PROGRAM AutoPreparationCtrl
VAR

	TON1: TON;
	TON2: TON;
	TON3: TON;
	TON4: TON;
	TON5: TON;
	TON6: TON;
	TON7: TON;
	TON8: TON;
	TON9: TON;
	TON10: TON;
	TON11: TON;
	TON12: TON;
	TON13: TON;
	TON14: TON;
	TON15: TON;
	TON16: TON;

	PreparationBypassTimer: TON;
	bPreparationBypassEn : BOOL;

	ARfbStnDegassCtrl: ARRAY [1..iStnQty] OF fbStnDegassCtrl;

	ARbStnDegassInProcess: ARRAY [1..iStnQty] OF BOOL;

	tStn1IncomingValveDelayOn: TON;
	tStn1aIncomingValveDelayOn: TON;
	tStn2IncomingValveDelayOn: TON;
	tStn3IncomingValveDelayOn: TON;
	tStn5IncomingValveDelayOn: TON;

	bA1PnpStep6: BOOL;
END_VAR
VAR // added by the converter: edge detectors and wires of the graphical bodies
    _w1 : BOOL;
END_VAR

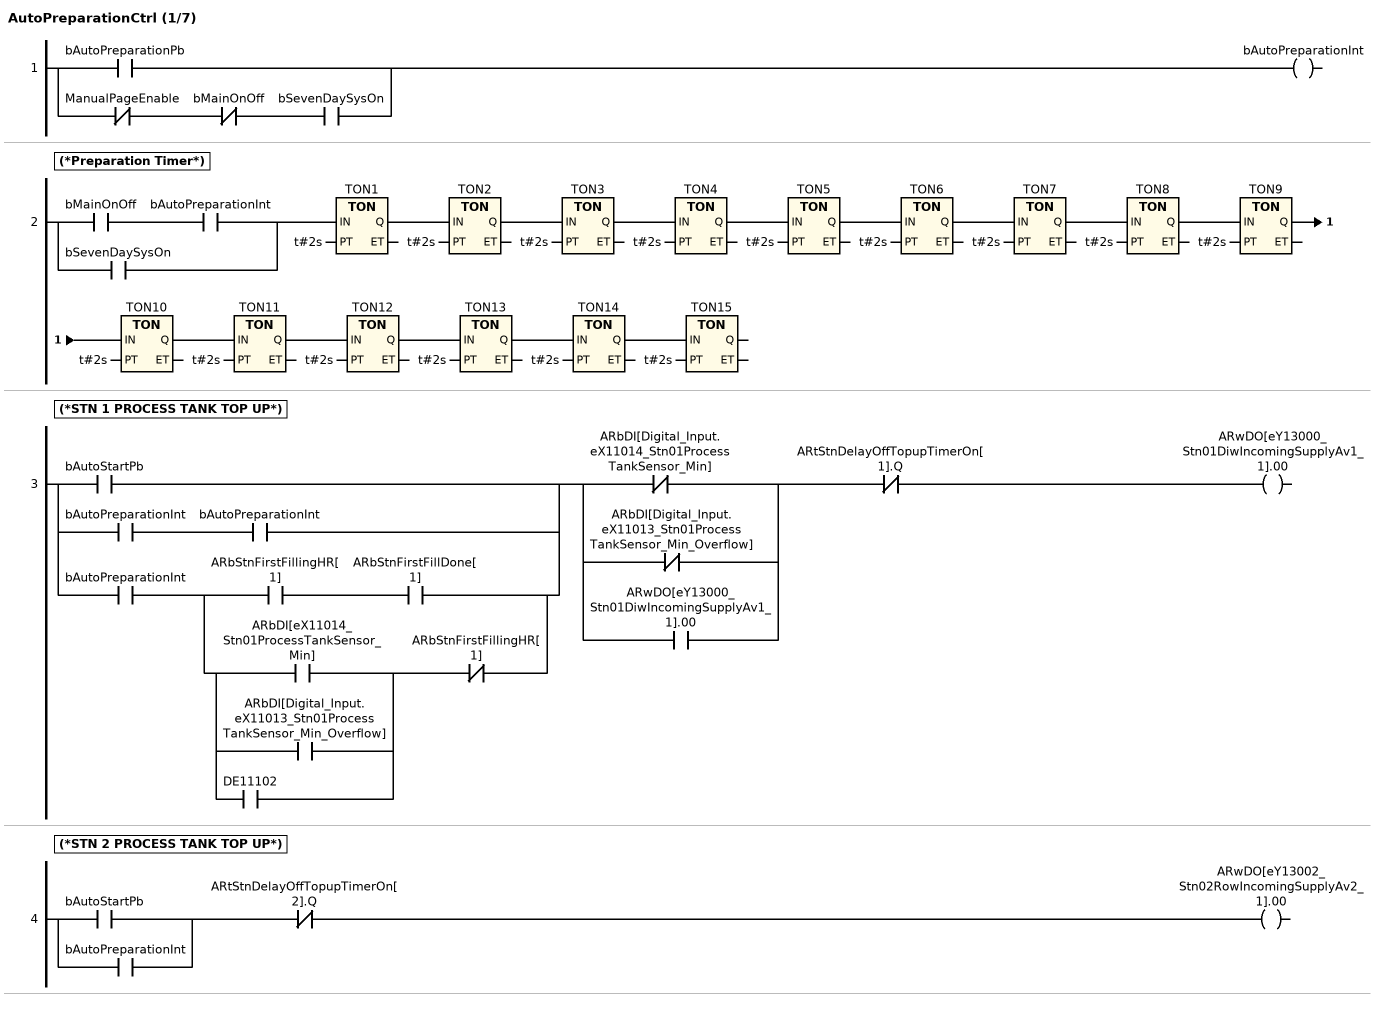
// NETWORK 1
bAutoPreparationInt := bAutoPreparationPb OR NOT ManualPageEnable AND NOT bMainOnOff AND bSevenDaySysOn;

// NETWORK 2
// label: (*Preparation Timer*)
TON1(IN := bMainOnOff AND bAutoPreparationInt OR bSevenDaySysOn, PT := t#2s); // TON
TON2(IN := TON1.Q, PT := t#2s); // TON
TON3(IN := TON2.Q, PT := t#2s); // TON
TON4(IN := TON3.Q, PT := t#2s); // TON
TON5(IN := TON4.Q, PT := t#2s); // TON
TON6(IN := TON5.Q, PT := t#2s); // TON
TON7(IN := TON6.Q, PT := t#2s); // TON
TON8(IN := TON7.Q, PT := t#2s); // TON
TON9(IN := TON8.Q, PT := t#2s); // TON
TON10(IN := TON9.Q, PT := t#2s); // TON
TON11(IN := TON10.Q, PT := t#2s); // TON
TON12(IN := TON11.Q, PT := t#2s); // TON
TON13(IN := TON12.Q, PT := t#2s); // TON
TON14(IN := TON13.Q, PT := t#2s); // TON
TON15(IN := TON14.Q, PT := t#2s); // TON

// NETWORK 3
// label: (*STN 1 PROCESS TANK TOP UP*)
ARwDO[eY13000_Stn01DiwIncomingSupplyAv1_1].00 := (bAutoStartPb OR bAutoPreparationInt AND bAutoPreparationInt OR bAutoPreparationInt AND (ARbStnFirstFillingHR[1] AND ARbStnFirstFillDone[1] OR (ARbDI[eX11014_Stn01ProcessTankSensor_Min] OR ARbDI[Digital_Input.eX11013_Stn01ProcessTankSensor_Min_Overflow] OR DE11102) AND NOT ARbStnFirstFillingHR[1])) AND (NOT ARbDI[Digital_Input.eX11014_Stn01ProcessTankSensor_Min] OR NOT ARbDI[Digital_Input.eX11013_Stn01ProcessTankSensor_Min_Overflow] OR ARwDO[eY13000_Stn01DiwIncomingSupplyAv1_1].00) AND NOT ARtStnDelayOffTopupTimerOn[1].Q;

// NETWORK 4
// label: (*STN 2 PROCESS TANK TOP UP*)
ARwDO[eY13002_Stn02RowIncomingSupplyAv2_1].00 := (bAutoStartPb OR bAutoPreparationInt) AND NOT ARtStnDelayOffTopupTimerOn[2].Q;

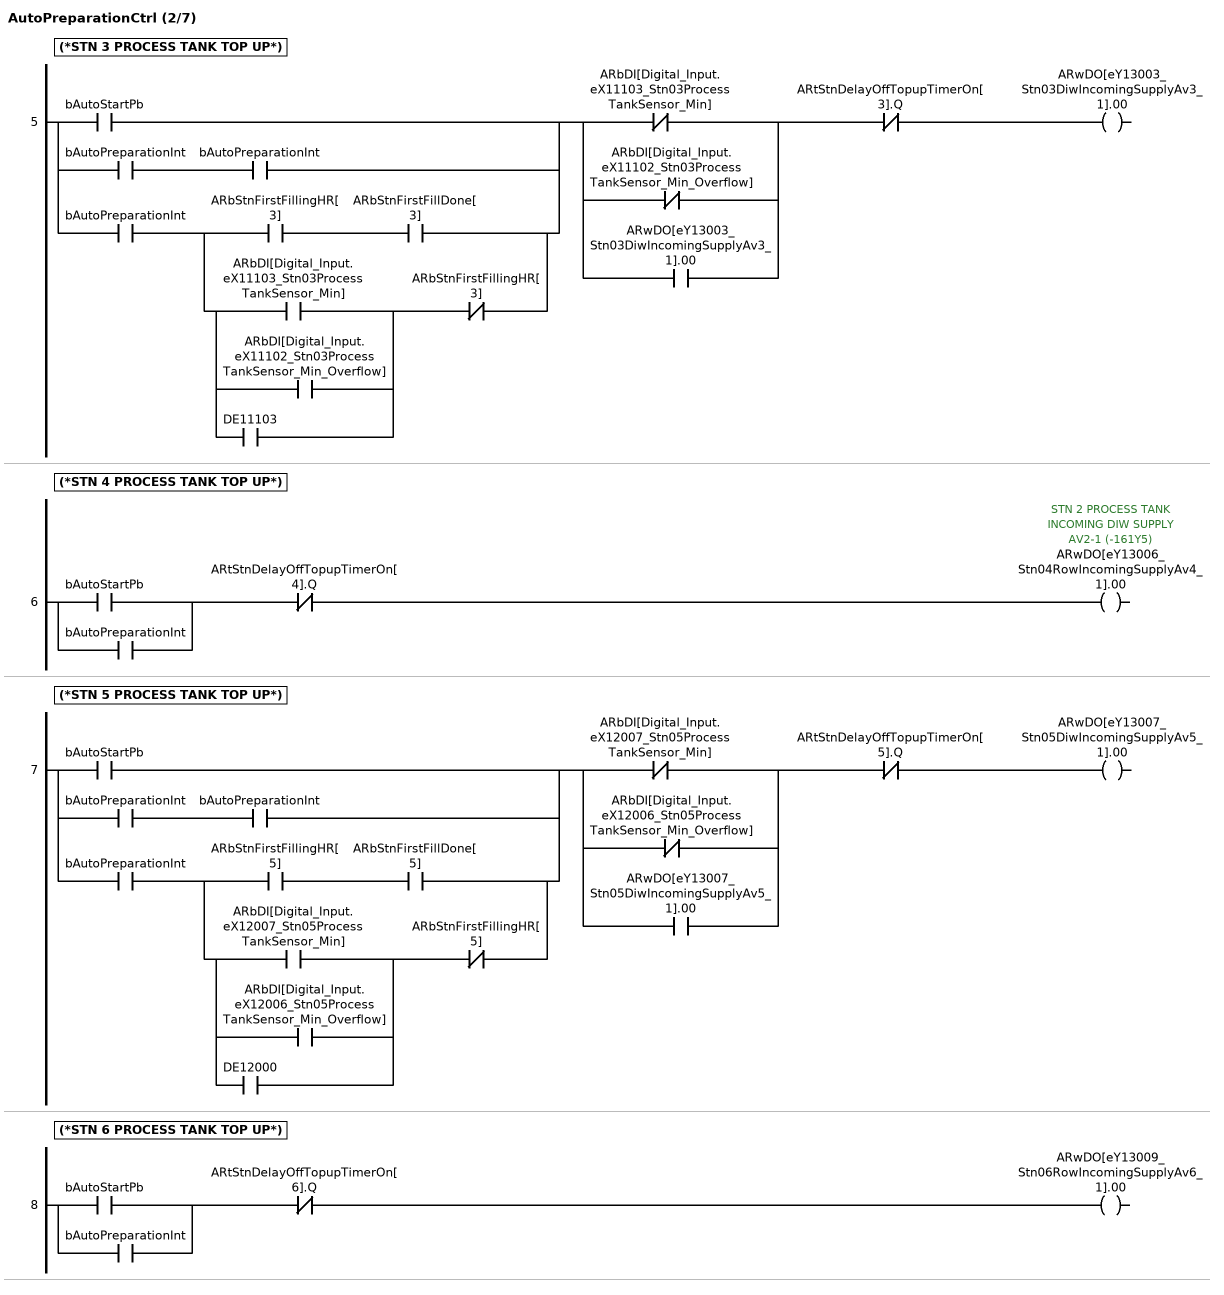
// NETWORK 5
// label: (*STN 3 PROCESS TANK TOP UP*)
ARwDO[eY13003_Stn03DiwIncomingSupplyAv3_1].00 := (bAutoStartPb OR bAutoPreparationInt AND bAutoPreparationInt OR bAutoPreparationInt AND (ARbStnFirstFillingHR[3] AND ARbStnFirstFillDone[3] OR (ARbDI[Digital_Input.eX11103_Stn03ProcessTankSensor_Min] OR ARbDI[Digital_Input.eX11102_Stn03ProcessTankSensor_Min_Overflow] OR DE11103) AND NOT ARbStnFirstFillingHR[3])) AND (NOT ARbDI[Digital_Input.eX11103_Stn03ProcessTankSensor_Min] OR NOT ARbDI[Digital_Input.eX11102_Stn03ProcessTankSensor_Min_Overflow] OR ARwDO[eY13003_Stn03DiwIncomingSupplyAv3_1].00) AND NOT ARtStnDelayOffTopupTimerOn[3].Q;

// NETWORK 6
//   ARwDO[eY13006_Stn04RowIncomingSupplyAv4_1].00: STN 2 PROCESS TANK INCOMING DIW SUPPLY AV2-1 (-161Y5)
// label: (*STN 4 PROCESS TANK TOP UP*)
ARwDO[eY13006_Stn04RowIncomingSupplyAv4_1].00 := (bAutoStartPb OR bAutoPreparationInt) AND NOT ARtStnDelayOffTopupTimerOn[4].Q;

// NETWORK 7
// label: (*STN 5 PROCESS TANK TOP UP*)
ARwDO[eY13007_Stn05DiwIncomingSupplyAv5_1].00 := (bAutoStartPb OR bAutoPreparationInt AND bAutoPreparationInt OR bAutoPreparationInt AND (ARbStnFirstFillingHR[5] AND ARbStnFirstFillDone[5] OR (ARbDI[Digital_Input.eX12007_Stn05ProcessTankSensor_Min] OR ARbDI[Digital_Input.eX12006_Stn05ProcessTankSensor_Min_Overflow] OR DE12000) AND NOT ARbStnFirstFillingHR[5])) AND (NOT ARbDI[Digital_Input.eX12007_Stn05ProcessTankSensor_Min] OR NOT ARbDI[Digital_Input.eX12006_Stn05ProcessTankSensor_Min_Overflow] OR ARwDO[eY13007_Stn05DiwIncomingSupplyAv5_1].00) AND NOT ARtStnDelayOffTopupTimerOn[5].Q;

// NETWORK 8
// label: (*STN 6 PROCESS TANK TOP UP*)
ARwDO[eY13009_Stn06RowIncomingSupplyAv6_1].00 := (bAutoStartPb OR bAutoPreparationInt) AND NOT ARtStnDelayOffTopupTimerOn[6].Q;

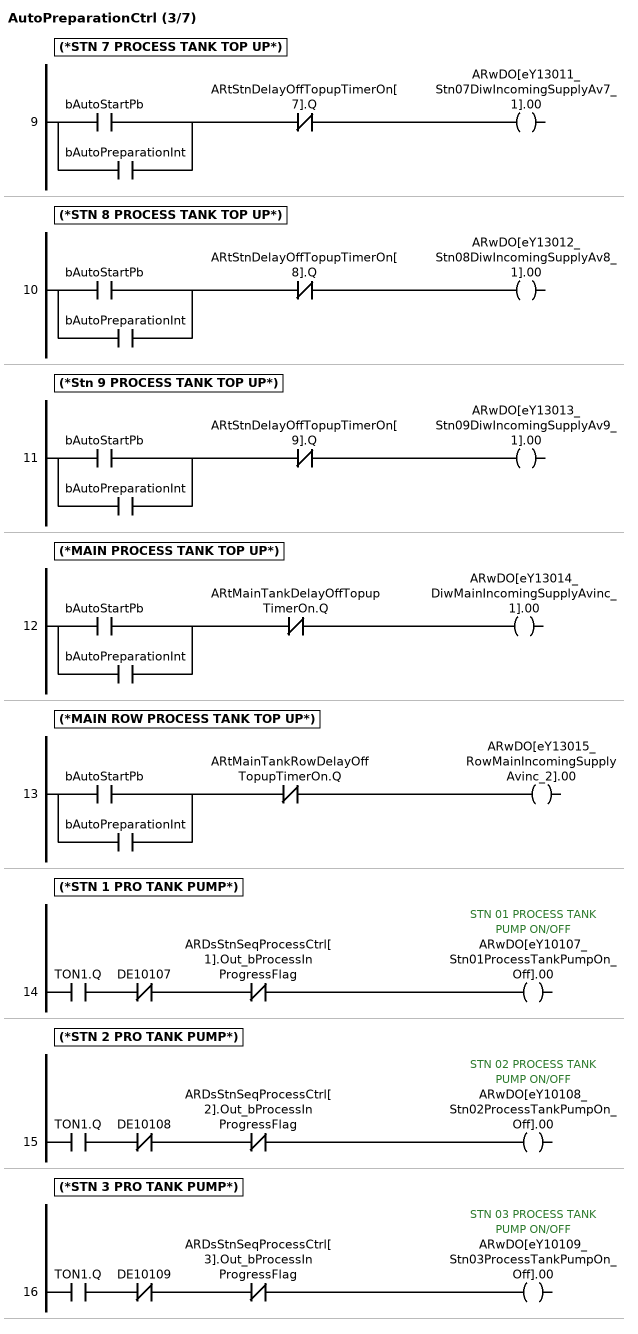
// NETWORK 9
// label: (*STN 7 PROCESS TANK TOP UP*)
ARwDO[eY13011_Stn07DiwIncomingSupplyAv7_1].00 := (bAutoStartPb OR bAutoPreparationInt) AND NOT ARtStnDelayOffTopupTimerOn[7].Q;

// NETWORK 10
// label: (*STN 8 PROCESS TANK TOP UP*)
ARwDO[eY13012_Stn08DiwIncomingSupplyAv8_1].00 := (bAutoStartPb OR bAutoPreparationInt) AND NOT ARtStnDelayOffTopupTimerOn[8].Q;

// NETWORK 11
// label: (*Stn 9 PROCESS TANK TOP UP*)
ARwDO[eY13013_Stn09DiwIncomingSupplyAv9_1].00 := (bAutoStartPb OR bAutoPreparationInt) AND NOT ARtStnDelayOffTopupTimerOn[9].Q;

// NETWORK 12
// label: (*MAIN PROCESS TANK TOP UP*)
ARwDO[eY13014_DiwMainIncomingSupplyAvinc_1].00 := (bAutoStartPb OR bAutoPreparationInt) AND NOT ARtMainTankDelayOffTopupTimerOn.Q;

// NETWORK 13
// label: (*MAIN ROW PROCESS TANK TOP UP*)
ARwDO[eY13015_RowMainIncomingSupplyAvinc_2].00 := (bAutoStartPb OR bAutoPreparationInt) AND NOT ARtMainTankRowDelayOffTopupTimerOn.Q;

// NETWORK 14
//   ARwDO[eY10107_Stn01ProcessTankPumpOn_Off].00: STN 01 PROCESS TANK PUMP ON/OFF
// label: (*STN 1 PRO TANK PUMP*)
ARwDO[eY10107_Stn01ProcessTankPumpOn_Off].00 := TON1.Q AND NOT DE10107 AND NOT ARDsStnSeqProcessCtrl[1].Out_bProcessInProgressFlag;

// NETWORK 15
//   ARwDO[eY10108_Stn02ProcessTankPumpOn_Off].00: STN 02 PROCESS TANK PUMP ON/OFF
// label: (*STN 2 PRO TANK PUMP*)
ARwDO[eY10108_Stn02ProcessTankPumpOn_Off].00 := TON1.Q AND NOT DE10108 AND NOT ARDsStnSeqProcessCtrl[2].Out_bProcessInProgressFlag;

// NETWORK 16
//   ARwDO[eY10109_Stn03ProcessTankPumpOn_Off].00: STN 03 PROCESS TANK PUMP ON/OFF
// label: (*STN 3 PRO TANK PUMP*)
ARwDO[eY10109_Stn03ProcessTankPumpOn_Off].00 := TON1.Q AND NOT DE10109 AND NOT ARDsStnSeqProcessCtrl[3].Out_bProcessInProgressFlag;

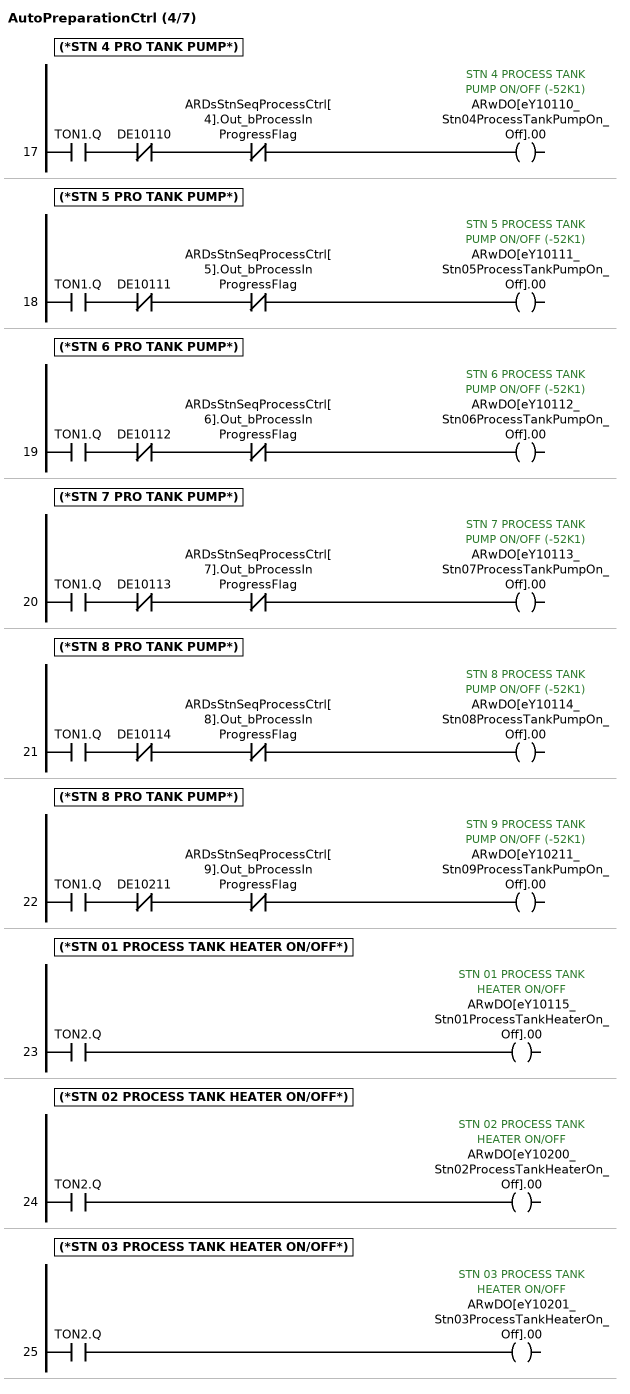
// NETWORK 17
//   ARwDO[eY10110_Stn04ProcessTankPumpOn_Off].00: STN 4 PROCESS TANK PUMP ON/OFF (-52K1)
// label: (*STN 4 PRO TANK PUMP*)
ARwDO[eY10110_Stn04ProcessTankPumpOn_Off].00 := TON1.Q AND NOT DE10110 AND NOT ARDsStnSeqProcessCtrl[4].Out_bProcessInProgressFlag;

// NETWORK 18
//   ARwDO[eY10111_Stn05ProcessTankPumpOn_Off].00: STN 5 PROCESS TANK PUMP ON/OFF (-52K1)
// label: (*STN 5 PRO TANK PUMP*)
ARwDO[eY10111_Stn05ProcessTankPumpOn_Off].00 := TON1.Q AND NOT DE10111 AND NOT ARDsStnSeqProcessCtrl[5].Out_bProcessInProgressFlag;

// NETWORK 19
//   ARwDO[eY10112_Stn06ProcessTankPumpOn_Off].00: STN 6 PROCESS TANK PUMP ON/OFF (-52K1)
// label: (*STN 6 PRO TANK PUMP*)
ARwDO[eY10112_Stn06ProcessTankPumpOn_Off].00 := TON1.Q AND NOT DE10112 AND NOT ARDsStnSeqProcessCtrl[6].Out_bProcessInProgressFlag;

// NETWORK 20
//   ARwDO[eY10113_Stn07ProcessTankPumpOn_Off].00: STN 7 PROCESS TANK PUMP ON/OFF (-52K1)
// label: (*STN 7 PRO TANK PUMP*)
ARwDO[eY10113_Stn07ProcessTankPumpOn_Off].00 := TON1.Q AND NOT DE10113 AND NOT ARDsStnSeqProcessCtrl[7].Out_bProcessInProgressFlag;

// NETWORK 21
//   ARwDO[eY10114_Stn08ProcessTankPumpOn_Off].00: STN 8 PROCESS TANK PUMP ON/OFF (-52K1)
// label: (*STN 8 PRO TANK PUMP*)
ARwDO[eY10114_Stn08ProcessTankPumpOn_Off].00 := TON1.Q AND NOT DE10114 AND NOT ARDsStnSeqProcessCtrl[8].Out_bProcessInProgressFlag;

// NETWORK 22
//   ARwDO[eY10211_Stn09ProcessTankPumpOn_Off].00: STN 9 PROCESS TANK PUMP ON/OFF (-52K1)
// label: (*STN 8 PRO TANK PUMP*)
ARwDO[eY10211_Stn09ProcessTankPumpOn_Off].00 := TON1.Q AND NOT DE10211 AND NOT ARDsStnSeqProcessCtrl[9].Out_bProcessInProgressFlag;

// NETWORK 23
//   ARwDO[eY10115_Stn01ProcessTankHeaterOn_Off].00: STN 01 PROCESS TANK HEATER ON/OFF
// label: (*STN 01 PROCESS TANK HEATER ON/OFF*)
ARwDO[eY10115_Stn01ProcessTankHeaterOn_Off].00 := TON2.Q;

// NETWORK 24
//   ARwDO[eY10200_Stn02ProcessTankHeaterOn_Off].00: STN 02 PROCESS TANK HEATER ON/OFF
// label: (*STN 02 PROCESS TANK HEATER ON/OFF*)
ARwDO[eY10200_Stn02ProcessTankHeaterOn_Off].00 := TON2.Q;

// NETWORK 25
//   ARwDO[eY10201_Stn03ProcessTankHeaterOn_Off].00: STN 03 PROCESS TANK HEATER ON/OFF
// label: (*STN 03 PROCESS TANK HEATER ON/OFF*)
ARwDO[eY10201_Stn03ProcessTankHeaterOn_Off].00 := TON2.Q;

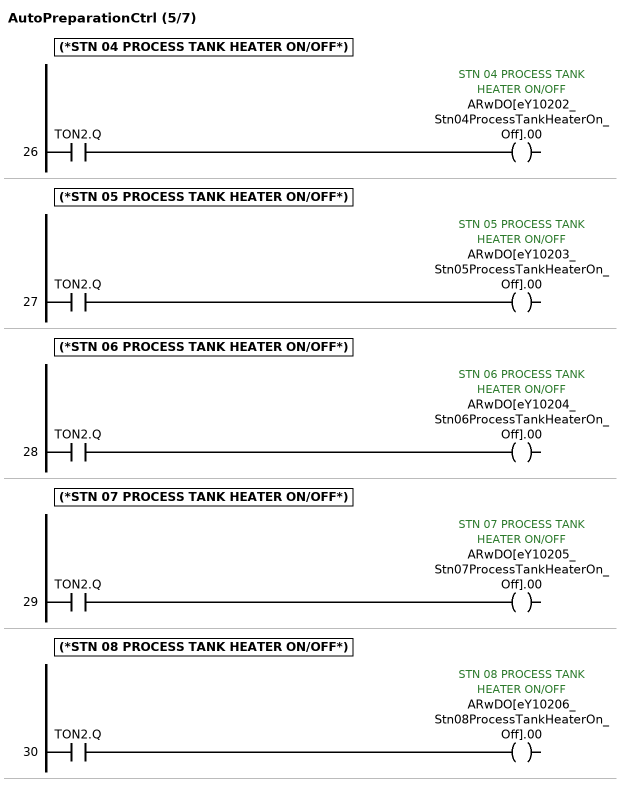
// NETWORK 26
//   ARwDO[eY10202_Stn04ProcessTankHeaterOn_Off].00: STN 04 PROCESS TANK HEATER ON/OFF
// label: (*STN 04 PROCESS TANK HEATER ON/OFF*)
ARwDO[eY10202_Stn04ProcessTankHeaterOn_Off].00 := TON2.Q;

// NETWORK 27
//   ARwDO[eY10203_Stn05ProcessTankHeaterOn_Off].00: STN 05 PROCESS TANK HEATER ON/OFF
// label: (*STN 05 PROCESS TANK HEATER ON/OFF*)
ARwDO[eY10203_Stn05ProcessTankHeaterOn_Off].00 := TON2.Q;

// NETWORK 28
//   ARwDO[eY10204_Stn06ProcessTankHeaterOn_Off].00: STN 06 PROCESS TANK HEATER ON/OFF
// label: (*STN 06 PROCESS TANK HEATER ON/OFF*)
ARwDO[eY10204_Stn06ProcessTankHeaterOn_Off].00 := TON2.Q;

// NETWORK 29
//   ARwDO[eY10205_Stn07ProcessTankHeaterOn_Off].00: STN 07 PROCESS TANK HEATER ON/OFF
// label: (*STN 07 PROCESS TANK HEATER ON/OFF*)
ARwDO[eY10205_Stn07ProcessTankHeaterOn_Off].00 := TON2.Q;

// NETWORK 30
//   ARwDO[eY10206_Stn08ProcessTankHeaterOn_Off].00: STN 08 PROCESS TANK HEATER ON/OFF
// label: (*STN 08 PROCESS TANK HEATER ON/OFF*)
ARwDO[eY10206_Stn08ProcessTankHeaterOn_Off].00 := TON2.Q;

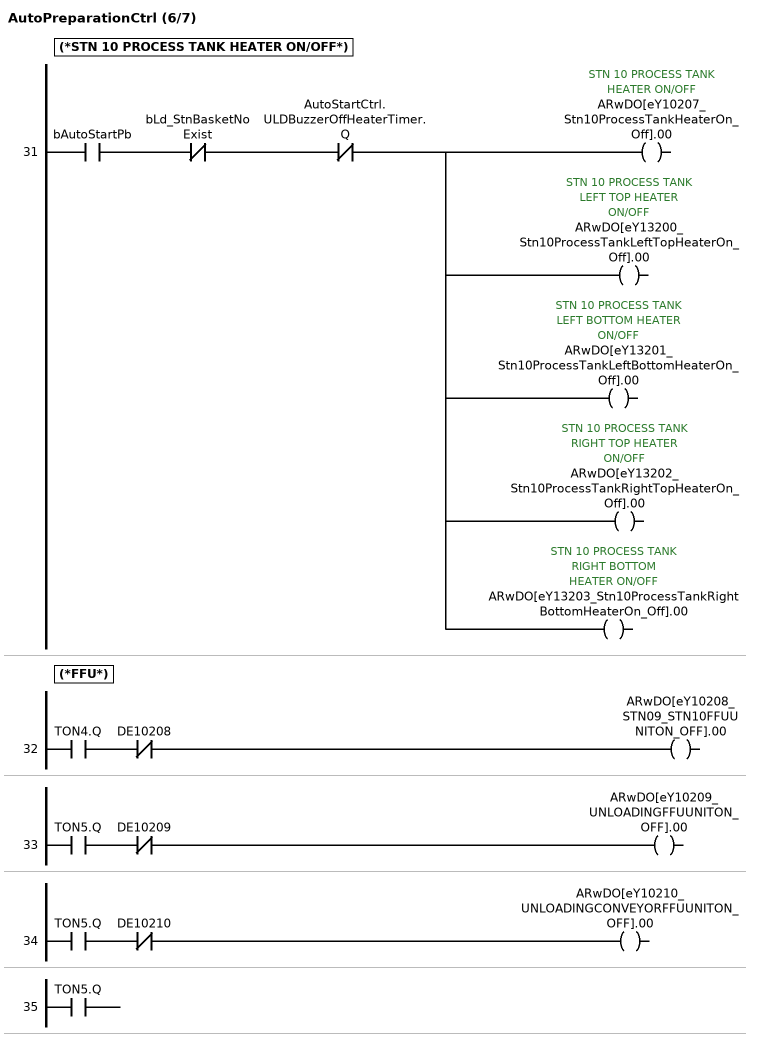
// NETWORK 31
//   ARwDO[eY10207_Stn10ProcessTankHeaterOn_Off].00: STN 10 PROCESS TANK HEATER ON/OFF
//   ARwDO[eY13200_Stn10ProcessTankLeftTopHeaterOn_Off].00: STN 10 PROCESS TANK LEFT TOP HEATER ON/OFF
//   ARwDO[eY13201_Stn10ProcessTankLeftBottomHeaterOn_Off].00: STN 10 PROCESS TANK LEFT BOTTOM HEATER ON/OFF
//   ARwDO[eY13202_Stn10ProcessTankRightTopHeaterOn_Off].00: STN 10 PROCESS TANK RIGHT TOP HEATER ON/OFF
//   ARwDO[eY13203_Stn10ProcessTankRightBottomHeaterOn_Off].00: STN 10 PROCESS TANK RIGHT BOTTOM HEATER ON/OFF
// label: (*STN 10 PROCESS TANK HEATER ON/OFF*)
_w1 := bAutoStartPb AND NOT bLd_StnBasketNoExist AND NOT AutoStartCtrl.ULDBuzzerOffHeaterTimer.Q;
ARwDO[eY10207_Stn10ProcessTankHeaterOn_Off].00 := _w1;
ARwDO[eY13200_Stn10ProcessTankLeftTopHeaterOn_Off].00 := _w1;
ARwDO[eY13201_Stn10ProcessTankLeftBottomHeaterOn_Off].00 := _w1;
ARwDO[eY13202_Stn10ProcessTankRightTopHeaterOn_Off].00 := _w1;
ARwDO[eY13203_Stn10ProcessTankRightBottomHeaterOn_Off].00 := _w1;

// NETWORK 32
// label: (*FFU*)
ARwDO[eY10208_STN09_STN10FFUUNITON_OFF].00 := TON4.Q AND NOT DE10208;

// NETWORK 33
ARwDO[eY10209_UNLOADINGFFUUNITON_OFF].00 := TON5.Q AND NOT DE10209;

// NETWORK 34
ARwDO[eY10210_UNLOADINGCONVEYORFFUUNITON_OFF].00 := TON5.Q AND NOT DE10210;

// NETWORK 35
(* TON5.Q; not connected *)

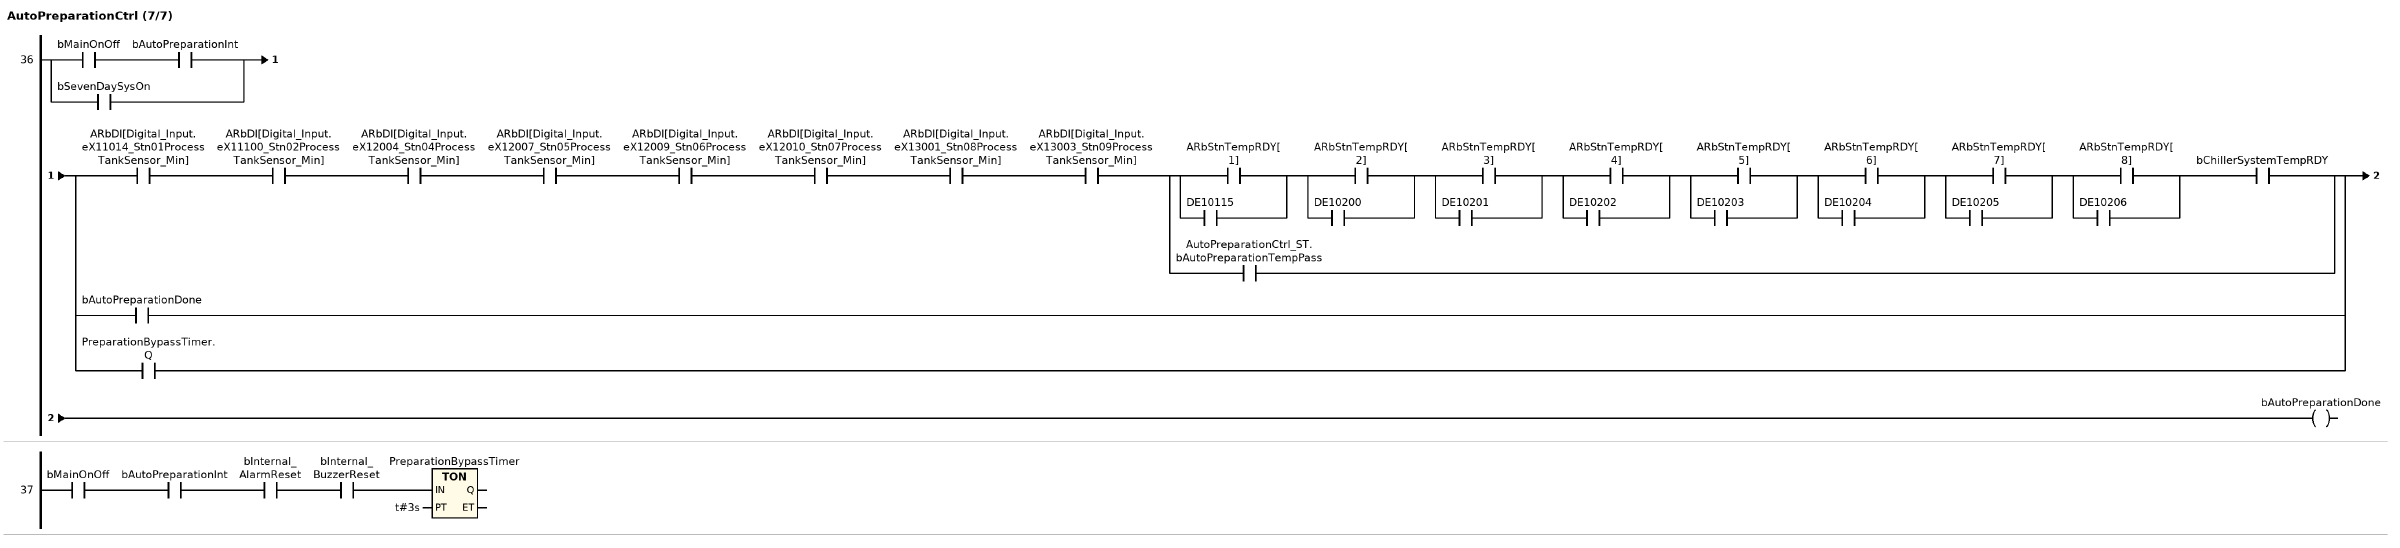
// NETWORK 36
bAutoPreparationDone := (bMainOnOff AND bAutoPreparationInt OR bSevenDaySysOn) AND (ARbDI[Digital_Input.eX11014_Stn01ProcessTankSensor_Min] AND ARbDI[Digital_Input.eX11100_Stn02ProcessTankSensor_Min] AND ARbDI[Digital_Input.eX12004_Stn04ProcessTankSensor_Min] AND ARbDI[Digital_Input.eX12007_Stn05ProcessTankSensor_Min] AND ARbDI[Digital_Input.eX12009_Stn06ProcessTankSensor_Min] AND ARbDI[Digital_Input.eX12010_Stn07ProcessTankSensor_Min] AND ARbDI[Digital_Input.eX13001_Stn08ProcessTankSensor_Min] AND ARbDI[Digital_Input.eX13003_Stn09ProcessTankSensor_Min] AND ((ARbStnTempRDY[1] OR DE10115) AND (ARbStnTempRDY[2] OR DE10200) AND (ARbStnTempRDY[3] OR DE10201) AND (ARbStnTempRDY[4] OR DE10202) AND (ARbStnTempRDY[5] OR DE10203) AND (ARbStnTempRDY[6] OR DE10204) AND (ARbStnTempRDY[7] OR DE10205) AND (ARbStnTempRDY[8] OR DE10206) AND bChillerSystemTempRDY OR AutoPreparationCtrl_ST.bAutoPreparationTempPass) OR bAutoPreparationDone OR PreparationBypassTimer.Q);

// NETWORK 37
PreparationBypassTimer(IN := bMainOnOff AND bAutoPreparationInt AND bInternal_AlarmReset AND bInternal_BuzzerReset, PT := t#3s); // TON

END_PROGRAM

(* stored: Version 1.1.0.1, ProductVersion 3.1.4024.11
   POU AutoPreparationCtrl: Id {c8b7667f-40dd-455a-b0f3-9e82d82c5b22}, SpecialFunc None *)
